FUNCTION INT_TO_SIZE : ST_SIZE
VAR_INPUT
	nValue : INT;
END_VAR

INT_TO_SIZE.nValue := INT_TO_UDINT(MAX(0, nValue));

END_FUNCTION

(* stored: Version 1.1.0.1, ProductVersion 3.1.4024.15
   POU INT_TO_SIZE: Id {59e07e0d-ac6f-4417-ab3c-899d72e40b38}, SpecialFunc None *)
